// TIA Portal V19 export
TYPE "LEXCHANGETRAY_typeHandlingXyzEm_toPlasticDeliver"
// stored: Access Published
   STRUCT
      feedback : "LEXCHANGETRAY_typeHandlingXyzEm_toPlasticFeedback";
      req : "LEXCHANGETRAY_typeHandlingXyzEm_toPlasticReq";
   END_STRUCT;
END_TYPE
